(* CODESYS project Results.library
   Company: _
   DefaultNamespace: Results
   Title: Results
   Placeholder: _Results
   Author: Krystian Lis et al.
   Description: Basic result implementation.
   Version: 1.0.0

Project tree, tasks and I/O mapping:
  libraries: Tc3_Module, * (Beckhoff Automation GmbH)
  Result/
    Error/
      global variables Err
      global variables GenericResult
    function IsErr [ST]
    function IsNone [ST]
    function IsNotNull [ST]
    function IsNull [ST]
    function IsOk [ST]
    function IsSome [ST]
    data type Result
*)

// Result/Result
TYPE Result : INT; END_TYPE

// Result/Error/Err
{attribute 'qualified_only'}
VAR_GLOBAL CONSTANT
	Itf0			: Result := -2;
	Str0			: Result := -3;
	ItfEq			: Result := -4;
	NoMatch			: Result := -5;
	Ptr0			: Result := -6;
	InvRef			: Result := -7;
	Ovf				: Result := -8;
	Udf				: Result := -9;
	Idx				: Result := -10;
	TcLib			: Result := -11;
	InfLoop			: Result := -12;
END_VAR

// Result/Error/GenericResult
VAR_GLOBAL CONSTANT
	None	: Result := 0;
	Ok		: Result := 1;
	Error	: Result := -1;
END_VAR

// Result/IsErr
FUNCTION IsErr : BOOL
VAR_INPUT
	eResult			: Result;
END_VAR
VAR_OUTPUT
	eCarry			: Result;
END_VAR

IsErr := eResult < 0;
eCarry := eResult;

END_FUNCTION

// Result/IsNone
FUNCTION IsNone : BOOL
VAR_INPUT
	eResult			: Result;
END_VAR
VAR_OUTPUT
	eCarry			: Result;
END_VAR

IsNone := eResult = 0;
eCarry := eResult;

END_FUNCTION

// Result/IsNotNull
FUNCTION IsNotNull : BOOL
VAR_INPUT
	anyPtrType		: ANY;
END_VAR

IF anyPtrType.diSize = SIZEOF(POINTER TO BYTE) THEN
	IsNotNull := anyPtrType.pValue^ <> 0;
END_IF

END_FUNCTION

// Result/IsNull
FUNCTION IsNull : BOOL
VAR_INPUT
	anyPtrType		: ANY;
END_VAR

IF anyPtrType.diSize = SIZEOF(POINTER TO BYTE) THEN
	IsNull := anyPtrType.pValue^ = 0;
END_IF

END_FUNCTION

// Result/IsOk
FUNCTION IsOk : BOOL
VAR_INPUT
	eResult			: Result;
END_VAR
VAR_OUTPUT
	eCarry			: Result;
END_VAR

IsOk := eResult > 0;
eCarry := eResult;

END_FUNCTION

// Result/IsSome
FUNCTION IsSome : BOOL
VAR_INPUT
	eResult			: Result;
END_VAR
VAR_OUTPUT
	eCarry			: Result;
END_VAR

IsSome := eResult <> 0;
eCarry := eResult;

END_FUNCTION
